// TIA Portal V16 export
// export: Created 2023-03-29T11:03:45.1101779Z, ExportSetting WithDefaults, DisplayName Totally Integrated Automation Portal, DisplayVersion V16 Update 6, DisplayName TIA Portal Version Control Interface, DisplayVersion V16 Update 2, DisplayName TIA Portal Openness, DisplayVersion V16 Update 6, DisplayName STEP 7 Professional, DisplayVersion V16 Update 6, DisplayName STEP 7 Safety, DisplayVersion V16, DisplayName WinCC Advanced, DisplayVersion V16 Update 6
VAR_GLOBAL   // PLC tag table "Z7"
   inputAumagotowośćZ_7 AT %M67.0 : Bool;   // znacznik wejście
   Hbit_Otwórz_Z7 AT %M22.4 : Bool;
   inputAwariaMomentZ_7 AT %M66.5 : Bool;   // znacznik wejście
   setAlarm_Moment_Z_7 AT %M67.4 : Bool;   // znacznik alarmu od momentówki w trybie zdalnym (aut/mamnual)
   isAUMA_Z_7 AT %M44.1 : Bool;   // przęłącznik wymiany na AUMA
   Hbit_Zamknieta_Z7 AT %M22.3 : Bool;
   Byte_Status_Z7 AT %MW22 : Word;   // Słowo statusu napędu
   CMD_Open_Z_7 AT %M67.5 : Bool;   // załącz otwieranie
   inputOtwartaZ_7 AT %M66.2 : Bool;   // znacznik wejście
   inputREMT_Z_7 AT %M66.1 : Bool;   // znacznik wejście zdalne
   inputAumaautomatZ_7 AT %M66.7 : Bool;   // znacznik wejście
   Hbit_Alarm_Z7 AT %M22.0 : Bool;
   CMD_Close_Z_7 AT %M67.6 : Bool;   // załącz zamykanie
   inputRuch_Z_7 AT %M66.4 : Bool;
   setSVMC_Z_7 AT %M67.3 : Bool;   // Znacznik polecenia zamknij w trybie automat
   setSVMO_Z_7 AT %M67.2 : Bool;   // Znacznik polecenia otwórz w trybie automat
   Hbit_Auto_Manu_Z7 AT %M22.7 : Bool;
   inputAumaawariaZ_7 AT %M67.1 : Bool;   // znacznik wejście
   CMD_Awaria_Z_7 AT %M67.7 : Bool;   // Awaria zbiorcza
   inputAumalokalneZ_7 AT %M66.6 : Bool;   // znacznik wejście
   Hbit_Reset_Z7 AT %M22.6 : Bool;
   isGotowość_Z_7 AT %M66.0 : Bool;   // bit gotowości wspólny
   Hbit_Otwarta_Z7 AT %M22.1 : Bool;
   Hbit_Zamknij_Z7 AT %M22.5 : Bool;
   inputZamkniętaZ_7 AT %M66.3 : Bool;   // znacznik wejście
   Hbit_REN_Z7 AT %M22.2 : Bool;
END_VAR
